// TwinCAT 3 PLC project RotaryPLC
// ProgramVersion: 3.1.4026.22
// libraries:
//   Tc2_MC2, * (Beckhoff Automation GmbH)
//   Tc2_Standard, * (Beckhoff Automation GmbH)
//   Tc2_System, * (Beckhoff Automation GmbH)
//   Tc3_EventLogger, * (Beckhoff Automation GmbH)
//   Tc3_IotBase, * (Beckhoff Automation GmbH)
//   TcUnit, * (www.tcunit.org)
// project tree:
//   DUTs/ E_MachineState.TcDUT
//   GVLs/ GVL_Motion.TcGVL, GVL_Safety.TcGVL
//   / PlcTask.TcTTO
//   POUs/01_Interfaces/ I_DigitalSensor.TcIO, I_Drive.TcIO
//   POUs/02_Hardware_Wrappers/ FB_DigitalSensor.TcPOU, FB_Drive.TcPOU
//   POUs/03_Modules/ FB_InfeedConveyor.TcPOU, FB_RotaryKnife.TcPOU
//   POUs/04_Machine_Logic/ FB_MainMachine.TcPOU
//   POUs/05_Tests/ FB_DigitalSensor_Test.TcPOU, FB_MainMachine_Test.TcPOU, PRG_TESTS.TcPOU
//   POUs/06_IoT_Edge/ FB_Telemetry.TcPOU
//   POUs/ MAIN.TcPOU
// real-time tasks:
//   TASK PlcTask: cycle T#10ms, priority 20, ADS port 350
// motion (NC):

CONFIGURATION RotaryPLC
    RESOURCE PLC ON TwinCAT3
        TASK PlcTask(INTERVAL := T#10ms, PRIORITY := 20);
        PROGRAM MAIN WITH PlcTask : MAIN;
        PROGRAM PRG_TESTS WITH PlcTask : PRG_TESTS;
    END_RESOURCE
END_CONFIGURATION

// ---- DUTs/E_MachineState.TcDUT
{attribute 'qualified_only'}
{attribute 'strict'}
TYPE E_MachineState :
(
    UNDEFINED   := 0,
    
    // --- The 'Stop' States (Normal Operations) ---
    STOPPED     := 10,
    STARTING    := 20,
    EXECUTE     := 30,
    
    // --- The 'Pause' States (Minor Jams / Upstream Backup) ---
    HOLDING     := 40,
    HELD        := 50,
    UNHOLDING   := 60,
    
    // --- The 'Fault' States (Safety or Major Errors) ---
    ABORTING    := 70,   // Rapid safe stop
    ABORTED     := 80,   // Safe state reached
    CLEARING    := 90,   // Operator acknowledging faults
    
    // --- Custom / Auxiliary Modes ---
    CLEANING    := 100   // Washdown mode (Actuators disabled, but machine 'On')
);
END_TYPE

// ---- GVLs/GVL_Motion.TcGVL
{attribute 'qualified_only'}
VAR_GLOBAL
    // Real, persistent memory instances that the NC tree will bind to
    stConveyorAxis : AXIS_REF;
    stKnifeAxis    : AXIS_REF;
END_VAR

// ---- GVLs/GVL_Safety.TcGVL
{attribute 'qualified_only'}
VAR_GLOBAL
    // 1. Physical Hardware Input (e.g., from TwinSAFE logic terminals)
    bPhysicalSafetyOk AT %I* : BOOL;

    // 2. Simulation Hooks (Defaulted to TRUE so the portfolio runs instantly)
    bSimulationMode : BOOL := TRUE;
    bSimulateSafety : BOOL := TRUE;

    // 3. The final evaluated safety state used by the machine logic
    bSafetyOk : BOOL;
END_VAR

// ---- POUs/01_Interfaces/I_DigitalSensor.TcIO
INTERFACE I_DigitalSensor

PROPERTY P_FallingEdge : BOOL
GET
END_GET
END_PROPERTY

PROPERTY P_InvertLogic : BOOL
GET
END_GET
SET
END_SET
END_PROPERTY

PROPERTY P_IsActive : BOOL
GET
END_GET
END_PROPERTY

PROPERTY P_RawInput : BOOL
GET
END_GET
SET
END_SET
END_PROPERTY

PROPERTY P_RisingEdge : BOOL
GET
END_GET
END_PROPERTY

END_INTERFACE

// ---- POUs/01_Interfaces/I_Drive.TcIO
INTERFACE I_Drive

METHOD M_Home : BOOL
VAR_INPUT
END_VAR
END_METHOD

METHOD M_MoveAbs : BOOL
VAR_INPUT
    fPosition : LREAL; // Target position in mm or degrees
    fVelocity : LREAL; // Speed for this move
END_VAR
END_METHOD

METHOD M_MoveVelocity : BOOL
VAR_INPUT
    fVelocity   : LREAL;         // Target speed in mm/s
    nDirection  : MC_Direction;  // 1 = Positive, 2 = Negative, 3 = Current
END_VAR
END_METHOD

METHOD M_Reset : BOOL
VAR_INPUT
END_VAR
END_METHOD

METHOD M_Stop : BOOL
VAR_INPUT
END_VAR
END_METHOD

PROPERTY P_Axis : REFERENCE TO AXIS_REF
GET
END_GET
END_PROPERTY

PROPERTY P_Busy : BOOL
GET
END_GET
END_PROPERTY

PROPERTY P_Enabled : BOOL
GET
END_GET
SET
END_SET
END_PROPERTY

PROPERTY P_Error : BOOL
GET
END_GET
END_PROPERTY

PROPERTY P_Ready : BOOL
GET
END_GET
END_PROPERTY

END_INTERFACE

// ---- POUs/MAIN.TcPOU
PROGRAM MAIN
VAR
    // This is the single instance of our entire modular machine.
    // By keeping it here, we keep the global namespace perfectly clean.
	{attribute 'OPC.UA.DA' := '1'}
    RotaryCutter : FB_MainMachine;
END_VAR

// =========================================================
// 1. HARDWARE / SIMULATION MULTIPLEXER
// =========================================================
IF GVL_Safety.bSimulationMode THEN
    GVL_Safety.bSafetyOk := GVL_Safety.bSimulateSafety;
ELSE
    GVL_Safety.bSafetyOk := GVL_Safety.bPhysicalSafetyOk;
END_IF

// =========================================================
// 2. EXECUTE THE MACHINE
// =========================================================
RotaryCutter();

END_PROGRAM

// ---- POUs/04_Machine_Logic/FB_MainMachine.TcPOU
FUNCTION_BLOCK FB_MainMachine
VAR_INPUT
    // --- Operator Commands ---
    {attribute 'OPC.UA.DA' := '1'}
    bCmdStart       : BOOL;
    
    {attribute 'OPC.UA.DA' := '1'}
    bCmdStop        : BOOL;
    
    {attribute 'OPC.UA.DA' := '1'}
    bCmdReset       : BOOL;
END_VAR

VAR_OUTPUT
    // --- State Machine Tracking ---
    {attribute 'OPC.UA.DA' := '1'}
    eState          : E_MachineState := E_MachineState.STOPPED;
    
    {attribute 'OPC.UA.DA' := '1'}
    udiCutsCompleted : UDINT;
END_VAR

VAR
    // --- The Physical Modules (Private) ---
    InfeedConveyor  : FB_InfeedConveyor;
    RotaryKnife     : FB_RotaryKnife;
    
    // --- The Virtual Motors (Private) ---
    ConveyorMotor   : FB_Drive;
    KnifeMotor      : FB_Drive;

    // --- Concrete Hardware Instances for Simulation (Private) ---
    fbProductSensor : FB_DigitalSensor;
    
    // --- Edge/IoT Telemetry (Private) ---
    EdgeGateway     : FB_Telemetry;
    
    // --- Industrial Diagnostics (Alarms) (Private) ---
    fbEventLogger      : FB_TcEventLogger;
    fbAlarmJam         : FB_TcAlarm;      // Alarm for material jams
    fbAlarmSafety      : FB_TcAlarm;      // Alarm for E-Stop / Safety Trips
    bAlarmsInitialized : BOOL;            // Flag to run setup code only once
    tonSensorJam       : TON;             // Detects if material is stuck
    
    // --- Safety Interface (Private) ---
    bSafetyOk          : BOOL;            // Locally mapped safety signal
END_VAR

// =========================================================
// 0. SAFETY MONITORING
// =========================================================
bSafetyOk := GVL_Safety.bSafetyOk;

// If safety drops, force the state machine into the ABORT sequence immediately.
IF NOT bSafetyOk AND eState <> E_MachineState.ABORTING AND eState <> E_MachineState.ABORTED THEN
    eState := E_MachineState.ABORTING;
END_IF

// =========================================================
// 1. HARDWARE LINKING
// =========================================================
fbProductSensor.bSimulationMode := TRUE;
InfeedConveyor.iProductCam := fbProductSensor;
InfeedConveyor.iMotor      := ConveyorMotor;
RotaryKnife.iMotor         := KnifeMotor;

// =========================================================
// 2. THE PACKML STATE MACHINE
// =========================================================
CASE eState OF

    E_MachineState.UNDEFINED:
        eState := E_MachineState.STOPPED;

    // ---------------------------------------------------------
    // NORMAL OPERATIONS
    // ---------------------------------------------------------
    E_MachineState.STOPPED:
        IF bCmdStart AND bSafetyOk THEN
            bCmdStart := FALSE;
            eState := E_MachineState.STARTING;
        END_IF

    E_MachineState.STARTING:
        // Trigger the homing routine we built in Phase 1
        RotaryKnife.bHomeCommand := TRUE;
        
        // PHASE 2 FIX: Wait for homing to finish AND ensure no NC errors
        IF NOT RotaryKnife.iMotor.P_Busy AND NOT RotaryKnife.iMotor.P_Error THEN 
            RotaryKnife.bHomeCommand := FALSE;
            eState := E_MachineState.EXECUTE;
            
            // --- NEW: Print to console when machine starts ---
            ADSLOGSTR(msgCtrlMask := ADSLOG_MSGTYPE_HINT, msgFmtStr := '>>> MACHINE STARTED: Reached EXECUTE State <<<', strArg := '');
        END_IF

    E_MachineState.EXECUTE:
        RotaryKnife.bEnable := TRUE;
        InfeedConveyor.bEnable := TRUE; 

        // --- NEW: Run the Master Conveyor at a constant speed ---
        // Parameter 1: Velocity (e.g., 500 mm/sec)
        // Parameter 2: Direction (1 = Positive)
        ConveyorMotor.M_MoveVelocity(500.0, 1);

        // Ninja Chop Logic (We will replace this with Gearing soon, but keep it for now)
        IF fbProductSensor.P_RisingEdge THEN
            RotaryKnife.bSyncCommand := TRUE;
            ADSLOGSTR(msgCtrlMask := ADSLOG_MSGTYPE_HINT, msgFmtStr := '>>> C++ HANDSHAKE OK: Product Detected! <<<', strArg := '');
        END_IF
        
        IF fbProductSensor.P_FallingEdge THEN
            RotaryKnife.bSyncCommand := FALSE;
            udiCutsCompleted := udiCutsCompleted + 1;
        END_IF
        
        IF bCmdStop THEN
            bCmdStop := FALSE;
            eState := E_MachineState.HOLDING;
        END_IF
		
    // ---------------------------------------------------------
    // PAUSING (Non-critical stops)
    // ---------------------------------------------------------
    E_MachineState.HOLDING:
        RotaryKnife.bSyncCommand := FALSE;
        eState := E_MachineState.HELD;

    E_MachineState.HELD:
        IF bCmdStart AND bSafetyOk THEN
            bCmdStart := FALSE;
            eState := E_MachineState.UNHOLDING;
        END_IF

    E_MachineState.UNHOLDING:
        eState := E_MachineState.EXECUTE;

    // ---------------------------------------------------------
    // FAULTS & SAFETY 
    // ---------------------------------------------------------
    E_MachineState.ABORTING:
        // Drop logical commands
        RotaryKnife.bSyncCommand := FALSE;
        
        // PHASE 2 FIX: Active braking for process faults (e.g., Jam)
        // If safety is still OK, we use servo torque to brake rather than coasting
        IF bSafetyOk THEN
            ConveyorMotor.M_Stop();
            KnifeMotor.M_Stop();
        END_IF
        
        eState := E_MachineState.ABORTED;

    E_MachineState.ABORTED:
        // Wait for physical safety to return AND operator to press Reset
        IF bSafetyOk AND bCmdReset THEN
            bCmdReset := FALSE;
            eState := E_MachineState.CLEARING;
        END_IF

    E_MachineState.CLEARING:
        // Require explicit Acknowledge (Confirm) before clearing
        fbAlarmJam.Confirm(0);
        fbAlarmJam.Clear(0, TRUE);
        
        fbAlarmSafety.Confirm(0);
        fbAlarmSafety.Clear(0, TRUE);
        
        // PHASE 1 FIX: Clear physical NC Axis faults before restarting
        ConveyorMotor.M_Reset();
        KnifeMotor.M_Reset();
        
        eState := E_MachineState.STOPPED;

    // ---------------------------------------------------------
    // AUXILIARY MODES
    // ---------------------------------------------------------
    E_MachineState.CLEANING:
        IF bCmdStop THEN
            bCmdStop := FALSE;
            eState := E_MachineState.STOPPED;
        END_IF

END_CASE

// =========================================================
// 3. INDUSTRIAL DIAGNOSTICS (ALARM LOGIC)
// =========================================================
IF NOT bAlarmsInitialized THEN
    fbAlarmJam.CreateEx(TC_Events.MachineAlarms.ConveyorSensorJam, TRUE, 0);
    fbAlarmSafety.CreateEx(TC_Events.MachineAlarms.SafetyTrip, TRUE, 0); 
    bAlarmsInitialized := TRUE;
END_IF

// --- Jam Detection ---
tonSensorJam(IN := (fbProductSensor.bRawInput AND eState = E_MachineState.EXECUTE), PT := T#5S);

IF tonSensorJam.Q THEN
    fbAlarmJam.Raise(0);
    eState := E_MachineState.ABORTING; 
END_IF

// =========================================================
// 4. HARDWARE SAFETY MASK & DRIVE POWER
// =========================================================
IF bSafetyOk THEN
    // Provide power/enable to the servo drives
    ConveyorMotor.bEnableCmd := TRUE;
    KnifeMotor.bEnableCmd    := TRUE;
ELSE
    // Drop power and logical commands immediately if safety is breached
    ConveyorMotor.bEnableCmd := FALSE;
    KnifeMotor.bEnableCmd    := FALSE;
    
    RotaryKnife.bEnable      := FALSE;
    RotaryKnife.bSyncCommand := FALSE;
    InfeedConveyor.bEnable   := FALSE; 
END_IF

// =========================================================
// 5. ALWAYS CALL THE MODULES AND MOTORS
// =========================================================
fbProductSensor();

// Pass the global references into the VAR_IN_OUT variables here:
ConveyorMotor(Axis := GVL_Motion.stConveyorAxis);
KnifeMotor(Axis := GVL_Motion.stKnifeAxis);

InfeedConveyor();
RotaryKnife();

// =========================================================
// 6. TELEMETRY & CLOUD SYNC
// =========================================================
EdgeGateway(
    eCurrentState := eState,
    udiCutsCompleted := udiCutsCompleted
);

END_FUNCTION_BLOCK

// ---- POUs/03_Modules/FB_InfeedConveyor.TcPOU
FUNCTION_BLOCK FB_InfeedConveyor
VAR_INPUT
    iMotor          : I_Drive;
    iProductCam     : I_DigitalSensor;
    
    // --- NEW: Commands from Main Machine ---
    bEnable         : BOOL; // <--- ADD THIS LINE
    
    // --- Machine Parameters ---
    fTargetVelocity : LREAL := 100.0;
END_VAR
VAR
END_VAR

// The conveyor is very simple for now. 
// It just ensures the motor is enabled and running.
IF iMotor <> 0 THEN
    iMotor.P_Enabled := bEnable;
    
    // ADDED: The required nDirection parameter to satisfy the interface
    iMotor.M_MoveVelocity(fVelocity := fTargetVelocity, nDirection := 1);
END_IF

END_FUNCTION_BLOCK

// ---- POUs/03_Modules/FB_RotaryKnife.TcPOU
FUNCTION_BLOCK FB_RotaryKnife
VAR_IN_OUT
    // --- Strict Compile-Time Hardware Bindings ---
    MasterAxis : AXIS_REF;
    SlaveAxis  : AXIS_REF;
END_VAR
VAR_INPUT
    iMotor          : I_Drive;
    bEnable         : BOOL;
    bEngageGearing  : BOOL; 
    
    {attribute 'TcLinkTo' := '1'}
    bSyncCommand AT %Q* : BOOL;
    
    bHomeCommand    : BOOL;  
    fKnifeDiameter  : LREAL := 100.0; 
END_VAR
VAR
    fbGearIn        : MC_GearIn;
    fbGearOut       : MC_GearOut;
    rtHome          : R_TRIG; 
    
    bIsSynchronized : BOOL;
    bError          : BOOL;
END_VAR

// 1. Safety Check: Only run if a motor has been assigned
IF iMotor <> 0 THEN
    
    // 2. Control the Motor Power
    iMotor.P_Enabled := bEnable;
    bError := iMotor.P_Error;

    // =========================================================
    // 3. HOMING SEQUENCE
    // =========================================================
    rtHome(CLK := bHomeCommand);
    IF rtHome.Q THEN
        iMotor.M_Home(); 
    END_IF

    // =========================================================
    // 4. ELECTRONIC GEARING (Synchronization)
    // =========================================================
    // Command to Lock the Knife to the Conveyor
    fbGearIn(
        Master           := MasterAxis,
        Slave            := SlaveAxis, 
        Execute          := bEngageGearing, 
        RatioNumerator   := 1,
        RatioDenominator := 1,
        Acceleration     := 10000,
        Deceleration     := 10000
    );
    
    bIsSynchronized := fbGearIn.InGear;
    
    // Command to Unlock (Stop following)
    fbGearOut(
        Slave            := SlaveAxis,
        Execute          := NOT bEngageGearing AND bIsSynchronized 
    );
    
END_IF

END_FUNCTION_BLOCK

// ---- POUs/02_Hardware_Wrappers/FB_Drive.TcPOU
FUNCTION_BLOCK FB_Drive IMPLEMENTS I_Drive
VAR_IN_OUT
    Axis : AXIS_REF; 
END_VAR

VAR_INPUT
    // --- External Commands ---
    bEnableCmd  : BOOL; 
END_VAR

VAR
    // --- Standard PLCopen Motion Blocks ---
    fbPower     : MC_Power;
    fbReset     : MC_Reset;
    fbStop      : MC_Stop;
    fbMoveAbs   : MC_MoveAbsolute;
    fbMoveVel   : MC_MoveVelocity;
    fbHome      : MC_Home;
END_VAR

// 1. Always Update the Axis Status
Axis.ReadStatus();

// 2. Power Control (Torque on/off)
fbPower(
    Axis := Axis,
    Enable := bEnableCmd,
    Enable_Positive := bEnableCmd,
    Enable_Negative := bEnableCmd
);

// 3. Call the Motion Function Blocks
// Note: We call them here so they can process their internal state machines
fbReset(Axis := Axis);
fbStop(Axis := Axis);
fbMoveAbs(Axis := Axis);
fbMoveVel(Axis := Axis);
fbHome(Axis := Axis);

// =========================================================
// CORRECTED TRIGGER RESET LOGIC
// =========================================================
// The Execute signals are now only dropped once the NC block 
// finishes its operation. This ensures the FB state machines 
// complete their execution and accurately reflect P_Busy.

IF fbReset.Done OR fbReset.Error THEN
    fbReset.Execute := FALSE;
END_IF

IF fbStop.Done OR fbStop.CommandAborted OR fbStop.Error THEN
    fbStop.Execute := FALSE;
END_IF

IF fbMoveAbs.Done OR fbMoveAbs.CommandAborted OR fbMoveAbs.Error THEN
    fbMoveAbs.Execute := FALSE;
END_IF

IF fbMoveVel.CommandAborted OR fbMoveVel.Error THEN
    fbMoveVel.Execute := FALSE;
END_IF

IF fbHome.Done OR fbHome.CommandAborted OR fbHome.Error THEN
    fbHome.Execute := FALSE;
END_IF

METHOD M_Home : BOOL
// Trigger a rising edge on the internal home block
// Note: We use the default homing mode configured in the TwinCAT NC Axis
fbHome.bCalibrationCam := FALSE; 
fbHome.Execute := TRUE;

M_Home := TRUE;
END_METHOD

METHOD M_MoveAbs : BOOL
VAR_INPUT
	(* Target position in mm or degrees*)
	fPosition	: LREAL;
	(* Speed for this move*)
	fVelocity	: LREAL;
END_VAR
// Trigger a rising edge on the internal motion block
fbMoveAbs.Position := fPosition;
fbMoveAbs.Velocity := fVelocity;
fbMoveAbs.Execute := TRUE; 

M_MoveAbs := TRUE; // Return TRUE to show the command was received
END_METHOD

METHOD M_MoveVelocity : BOOL
VAR_INPUT
    fVelocity   : LREAL;         // Target speed in mm/s
    nDirection  : MC_Direction;  // 1 = Positive, 2 = Negative, 3 = Current
END_VAR
// Pass the inputs to the underlying PLCopen block
fbMoveVel.Velocity  := fVelocity;
fbMoveVel.Direction := nDirection;
fbMoveVel.Execute   := TRUE;

M_MoveVelocity := TRUE;
END_METHOD

METHOD M_Reset : BOOL
fbReset.Execute := TRUE; M_Reset := TRUE;
END_METHOD

METHOD M_Stop : BOOL
fbStop.Execute := TRUE; M_Stop := TRUE;
END_METHOD

PROPERTY P_Axis : REFERENCE TO AXIS_REF
GET
P_Axis REF= Axis; // This creates a 'link' to the real Axis variable
END_GET
END_PROPERTY

PROPERTY P_Busy : BOOL
GET
// The axis is busy if it is physically moving or if a move block is still active
P_Busy := Axis.Status.Moving OR fbMoveAbs.Busy OR fbMoveVel.Busy OR fbHome.Busy;
END_GET
END_PROPERTY

PROPERTY P_Enabled : BOOL
GET
P_Enabled := bEnableCmd;
END_GET
SET
bEnableCmd := P_Enabled;
END_SET
END_PROPERTY

PROPERTY P_Error : BOOL
GET
P_Error := Axis.Status.Error;
END_GET
END_PROPERTY

PROPERTY P_Ready : BOOL
GET
P_Ready := Axis.Status.Operational;
END_GET
END_PROPERTY

END_FUNCTION_BLOCK

// ---- POUs/02_Hardware_Wrappers/FB_DigitalSensor.TcPOU
FUNCTION_BLOCK FB_DigitalSensor IMPLEMENTS I_DigitalSensor
VAR_INPUT
    // The physical hardware terminal mapping
    bRawInput AT %I* : BOOL; 
    
    // NEW: HiL Simulation Hooks
    bSimulationMode  : BOOL; // TRUE = Ignore physical %I*, use bSimulationInput
    {attribute 'TcLinkTo' := '1'}
	bSimulationInput AT %I* : BOOL;
END_VAR
VAR
    // Internal State (Private)
    bActive         : BOOL;
    bEffectiveInput : BOOL; // Multiplexer output
    bInvert         : BOOL;
    
    // Edge Detection
    fbRisingEdge  : R_TRIG;
    fbFallingEdge : F_TRIG;
END_VAR

// =========================================================
// 1. HARDWARE VS. SIMULATION MULTIPLEXER
// =========================================================
IF bSimulationMode THEN
    bEffectiveInput := bSimulationInput; // Listen to Python Twin
ELSE
    bEffectiveInput := bRawInput;        // Listen to Physical IO Terminal
END_IF

// =========================================================
// 2. Handle Wiring Logic (Normally Open vs Normally Closed)
// =========================================================
IF bInvert THEN
    bActive := NOT bEffectiveInput;
ELSE
    bActive := bEffectiveInput;
END_IF

// =========================================================
// 3. Run the Edge Detection Blocks
// =========================================================
fbRisingEdge(CLK := bActive);
fbFallingEdge(CLK := bActive);

PROPERTY P_FallingEdge : BOOL
GET
P_FallingEdge := fbFallingEdge.Q;
END_GET
END_PROPERTY

PROPERTY P_InvertLogic : BOOL
GET
P_InvertLogic := bInvert;
END_GET
SET
bInvert := P_InvertLogic;
END_SET
END_PROPERTY

PROPERTY P_IsActive : BOOL
GET
P_IsActive := bActive;
END_GET
END_PROPERTY

PROPERTY P_RawInput : BOOL
GET
P_RawInput := bRawInput;
END_GET
SET
bRawInput := P_RawInput;
END_SET
END_PROPERTY

PROPERTY P_RisingEdge : BOOL
GET
P_RisingEdge := fbRisingEdge.Q;
END_GET
END_PROPERTY

END_FUNCTION_BLOCK

// ---- POUs/06_IoT_Edge/FB_Telemetry.TcPOU
FUNCTION_BLOCK FB_Telemetry
VAR_INPUT
    // The main machine will pass its current state in here
    eCurrentState : E_MachineState; 
    
    // NEW: Metric for production tracking
    udiCutsCompleted : UDINT;
END_VAR
VAR
    // The TwinCAT MQTT Client
    fbMqttClient  : FB_IotMqttClient;
    
    // Connection Settings
    bEnableMqtt   : BOOL := TRUE;
    sBrokerIp     : STRING(255) := 'broker.hivemq.com'; // Free public testing broker
    sTopic        : STRING(255) := 'sahil/portfolio/machine/status';
    
    // Payload generation
    sPayload      : STRING(255);
    fbTimer       : TON; // Timer to publish data every 2 seconds
    
    // NEW: String helpers for JSON formatting
    sStateStr     : STRING;
    sCutStr       : STRING;
END_VAR

// 1. Configure the Client
fbMqttClient.sHostName := sBrokerIp;
fbMqttClient.nHostPort := 8883; // UPDATED: Changed from 1883 to 8883 for Secure MQTTS

// (Note for Portfolio: In a real factory, we would link the TLS cert path here)
// fbMqttClient.stTLS.sCA := 'C:\TwinCAT\Certificates\ca.crt';

// 2. Keep the Client running in the background
fbMqttClient.Execute(bConnect := bEnableMqtt);

// 3. Timer: Trigger every 2 seconds
fbTimer(IN := NOT fbTimer.Q, PT := T#2S);

// 4. Publish Data
IF fbMqttClient.bConnected AND fbTimer.Q THEN
    
    // Convert numbers to strings first
    sStateStr := TO_STRING(eCurrentState);
    sCutStr   := TO_STRING(udiCutsCompleted);
    
    // Build an Industry 4.0 JSON string. 
    // Example output: {"State": 30, "CutsCompleted": 150}
    sPayload := CONCAT('{"State": ', sStateStr);
    sPayload := CONCAT(sPayload, ', "CutsCompleted": ');
    sPayload := CONCAT(sPayload, sCutStr);
    sPayload := CONCAT(sPayload, '}');
    
    // Send it to the cloud
    fbMqttClient.Publish(
        sTopic       := sTopic, 
        pPayload     := ADR(sPayload), 
        nPayloadSize := INT_TO_UDINT(LEN(sPayload)) + 1, 
        eQoS         := TcIotMqttQos.AtMostOnceDelivery, 
        bRetain      := FALSE, 
        bQueue       := FALSE
    );
    
END_IF

END_FUNCTION_BLOCK

// ---- POUs/05_Tests/PRG_TESTS.TcPOU
PROGRAM PRG_TESTS
VAR
    // We declare instances of our test suites here
    DigitalSensorTest : FB_DigitalSensor_Test;
    
    // NEW: Add the Main Machine test suite
    MainMachineTest   : FB_MainMachine_Test; 
END_VAR

// This is the master command that tells TcUnit to run all tests and print the results
TcUnit.RUN();

END_PROGRAM

// ---- POUs/05_Tests/FB_DigitalSensor_Test.TcPOU
FUNCTION_BLOCK FB_DigitalSensor_Test EXTENDS TcUnit.FB_TestSuite
VAR
    // The actual sensor we are going to test
    Sensor : FB_DigitalSensor;
END_VAR

// Call the test methods here
Test_RisingEdge();

METHOD Test_RisingEdge : REFERENCE TO FB_Test
VAR_INPUT
END_VAR
// 1. Tell TcUnit we are starting a specific test
TEST('Test_RisingEdge');

// 2. Cycle 1: Ensure the sensor starts clear (False)
Sensor.bRawInput := FALSE;
Sensor(); 

// 3. Cycle 2: A chicken arrives! (Input goes True)
// This creates the rising edge.
Sensor.bRawInput := TRUE;
Sensor(); 

// 4. Verification 1: Did the property trigger?
// AssertTrue will fail the test if the condition is not met.
AssertTrue(
    Condition := Sensor.P_RisingEdge,
    Message   := 'FAILED: Rising edge did not trigger when input went high!'
);

// 5. Cycle 3: The chicken is still blocking the sensor
// We run the block one more time. The rising edge should disappear.
Sensor();

// 6. Verification 2: Did it act like a one-shot?
AssertFalse(
    Condition := Sensor.P_RisingEdge,
    Message   := 'FAILED: Rising edge stayed true for more than one cycle!'
);

// 7. Tell TcUnit this test is complete
TEST_FINISHED();
END_METHOD

END_FUNCTION_BLOCK

// ---- POUs/05_Tests/FB_MainMachine_Test.TcPOU
FUNCTION_BLOCK FB_MainMachine_Test EXTENDS TcUnit.FB_TestSuite
VAR
    // The machine instance we are going to test
    Machine : FB_MainMachine;
END_VAR

// Call the test methods here
Test_HomingSecurity();

METHOD Test_HomingSecurity
VAR
END_VAR
TEST('Test_HomingSecurity');

// // 1. Setup Initial State
// GVL_Safety.bSafetyOk := TRUE;
// Machine.eState := E_MachineState.STOPPED;
// Machine.bCmdStart := TRUE;
// 
// // 2. Run Machine (Should transition to STARTING)
// Machine();
// 
// // 3. Drop Start Command & Inject Homing Error
// Machine.bCmdStart := FALSE;
// 
// // We simulate a physical drive failure by forcing the NC Axis Status
// Machine.KnifeMotor.Axis.Status.Error := TRUE;  // Fake an NC Error
// Machine.KnifeMotor.Axis.Status.Moving := FALSE; // Fake that the axis is no longer moving (Not Busy)
// 
// // 4. Run Machine again (It will evaluate the STARTING -> EXECUTE transition)
// Machine();
// 
// // 5. ASSERTION: It must remain in STARTING and NOT jump to EXECUTE
// AssertEquals_DINT(
//     Expected := E_MachineState.STARTING,
//     Actual := Machine.eState,
//     Message := 'Failed Phase 2 Security: Machine entered EXECUTE with an active NC Error!'
// );
// 
// TEST_FINISHED();
END_METHOD

END_FUNCTION_BLOCK
